Universal Robots PolyScope program: raw01_movej.urp

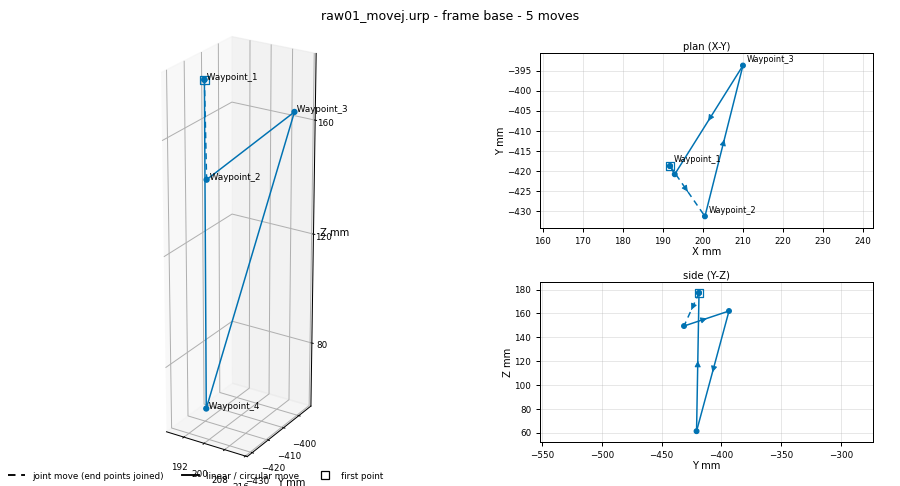
[picture p0: tool path of raw01_movej.urp in frame base, 5 of 5 moves have a stored position in this frame; points joined in program order, loops and branches not executed]
Program raw01_movej (installation=default directory=/programs createdIn=5.9.1.1031110 lastSavedIn=5.9.1.1031110 robotSerialNumber=20195501059)
Calibrated DH parameters: a=[0.000146, -0.418764, -0.053981, 0.000058, -0.000023, 0]; d=[0.162545, 37.319448, -206.067439, 168.881546, 0.09955, 0.099464]; alpha=[1.57004, -0.001979, 0.002304, 1.570607, -1.57066, 0]; deltaTheta=[0, -0.174616, -1.258233, 1.432844, -0.000001, 0]
Robot Program (runOnlyOnce=true)
  MoveJ speed 60 deg/s, acceleration 80 deg/s^2 (useActiveTCP=true) feature=Base
    Waypoint Waypoint_1: TCP in base x=191.775 y=-418.747 z=177.183 mm, rx=2.6851 ry=-0.62 rz=0.5262 rad; joints [87.655, -105.135, 137.507, -146.09, 287.063, -152.7] deg; TCP offset x=0 y=0 z=158 mm, rx=0 ry=0 rz=0 rad
    Waypoint Waypoint_2: TCP in base x=200.486 y=-431.303 z=149.488 mm, rx=2.685 ry=-0.6202 rz=0.5262 rad; joints [89.271, -99.116, 138.289, -153.337, 286.4, -151.139] deg
  MoveL speed 250 mm/s, acceleration 1200 mm/s^2 (useActiveTCP=true) feature=Base
    Waypoint Waypoint_3: TCP in base x=209.978 y=-393.65 z=162.057 mm, rx=2.6851 ry=-0.6201 rz=0.5261 rad; joints [91.051, -106.119, 141.044, -149.543, 285.674, -149.467] deg
    Waypoint Waypoint_4: TCP in base x=192.948 y=-420.801 z=61.457 mm, rx=3.0798 ry=-0.6201 rz=0 rad; joints [97.846, -82.651, 125.139, -132.481, 270.063, -149.346] deg
    MoveDirectionNode (selectedDirection=ZPlus toolParams=0.02, 1.2) feature=Joint_6_name
      Until TOOL_CONTACT_DETECTION (allowActions=false retraction=0.005 decelerationAcceleration=3 decelerationAngularAcceleration=34.906585)
    Waypoint Waypoint_1: TCP in base x=191.775 y=-418.747 z=177.183 mm, rx=2.6851 ry=-0.62 rz=0.5262 rad; joints [87.655, -105.135, 137.507, -146.09, 287.063, -152.7] deg
